(* CoDeSys 2.3 export: MIR_KOMPRESSOR.EXP *)

(* POU PLC_PRG, ST *)
PROGRAM PLC_PRG
VAR
	a : BOOL;
END_VAR
translate();
IF (_switchAuto) THEN
	work();
END_IF;
(*
start_or_stop(); *)
E_STOP();
END_PROGRAM

(* POU translate, ST *)
PROGRAM translate
VAR

	K3: BOOL;
	SC1: SCALE;
	SC2: SCALE;
	SC3: SCALE;
	SC4: SCALE;
	SC5: SCALE;
	SC6: SCALE;
	SC7: SCALE;
	SC8: SCALE;
	SC9: SCALE;
	SC10: SCALE;
	SC11: SCALE;
	SC12: SCALE;
END_VAR
MODBUS();
ANALOG();
K01 := TRM7;
K1 := _1pressLevelInDI;
K2 := _2pressLevelInDI;
K3 := _3pressLevelInDI;
K4 := _4pressLevelInDI;
 _rejimModeDO := P2;

IF (kompOnDO_MB = TRUE) THEN
	_kompOnDO :=  kompOnDO_MB;
ELSE
	_kompOnDO := FALSE;
END_IF;
IF (kompOffDO_MB = TRUE ) THEN
	_kompOffDO :=  kompOffDO_MB;
ELSE
	_kompOffDO := FALSE;
END_IF
END_PROGRAM
ACTION ANALOG:
SC1(IN := %IW0, MIN_VALUE := 4, MAX_VALUE := 20, OUT => analog1);
SC2(IN := %IW1, MIN_VALUE := 4, MAX_VALUE := 20, OUT => analog2);
SC3(IN := %IW2, MIN_VALUE := 4, MAX_VALUE := 20, OUT => analog3);
SC4(IN := %IW3, MIN_VALUE := 4, MAX_VALUE := 20, OUT => analog4);
SC5(IN := %IW4,MIN_VALUE := 4, MAX_VALUE := 20,  OUT => analog5);
SC6(IN := %IW5,MIN_VALUE := 4, MAX_VALUE := 20,  OUT => analog6);
SC7(IN := %IW6, MIN_VALUE := 4, MAX_VALUE := 20, OUT => analog7);
SC8(IN := %IW7, MIN_VALUE := 4, MAX_VALUE := 20, OUT => analog8);
SC9(IN := %IW8, MIN_VALUE := 4, MAX_VALUE := 20, OUT => analog9);
SC10(IN := %IW9, MIN_VALUE := 4, MAX_VALUE := 20, OUT => analog10);
SC11(IN := %IW10, MIN_VALUE := 4, MAX_VALUE := 20, OUT => analog11);
SC12(IN := %IW11, MIN_VALUE := 4, MAX_VALUE := 20, OUT => analog12);
END_ACTION
ACTION MODBUS:
S4_1MB := S4_1;
S4_2MB := S4_2;
S5_1MB := S5_1;
S5_2MB := S5_2;
S6_1MB := S6_1;
S6_2MB := S6_2;
S7_1MB := S7_1;
S7_2MB := S7_2;
S8_1MB := S8_1;
S8_2MB := S8_2;
S9_1MB := S9_1;
S9_2MB := S9_2;
S10_1MB := S10_1;
S10_2MB := S10_2;
S11_1MB := S11_1;
S11_2MB := S11_2;
S14_1MB := S14_1;
S14_2MB := S14_2;
S18_1MB := S18_1;
S18_2MB := S18_2;
S19_1MB := S19_1;
S19_2MB := S19_2;
controlFazaDIMB := _controlFazaDI;
currentHighJD5DIMB := _currentHighJD5DI;
vacumContactOnDIMB := _vacumContactOnDI;
press1LevelInDIMB := _1pressLevelInDI;
press2LevelInDIMB := _2pressLevelInDI;
press3LevelInDIMB := _3pressLevelInDI;
press4LevelInDIMB := _4pressLevelInDI;
press4LevelOutDIMB :=_4pressLeveOutDI;
pressWaterDIMB := _pressWaterDI;

KM4_1MB := KM4_1;
KM4_2MB := KM4_2;
KM5_1MB := KM5_1;
KM5_2MB := KM5_2;
KM6_1MB := KM6_1;
KM6_2MB := KM6_2;
KM7_1MB := KM7_1;
KM7_2MB := KM7_2;
KM8_1MB := KM8_1;
KM8_2MB := KM8_2;
KM9_1MB := KM9_1;
KM9_2MB := KM9_2;
KM10_1MB := KM10_1;
KM10_2MB := KM10_2;
KM11_1MB := KM11_1;
KM11_2MB := KM11_2;

KM14_1MB := KM14_1;
KM14_2MB := KM14_2;
KM18_1MB := KM18_1;
KM18_2MB := KM18_2;
KM19_1MB := KM19_1;
KM19_2MB := KM19_2;
KM1_MB := KM1;
KM2_MB := KM2;
(*
kompOnDO_MB := _kompOnDO;
kompOffDO_MB := _kompOffDO;*)
alarmLedDO_MB := _alarmLedDO;
stopModeDO_MB := _stopModeDO;

konsovikMechanikMotor := _konsovikMechanikMotor;
emergencyStop_MB := NOT _emergencyStop;
SBA41_MB := SBA41;
SB42_MB := SB42;
SB43_MB := SB43;
SB44_MB := SB44;
SB53_1MB := SB53_1;




buttonStop_MB := _buttonStop;
buttonRejim_MB := _buttonRejim;
buttonPusk_MB := _buttonPusk;
switchAuto_MB := _switchAuto;
switchManual_MB := _switchManual;
emergencyStopmashZal_MB := NOT  _emergencyStopMashZal;
END_ACTION

(* POU SCALE, ST *)
FUNCTION_BLOCK SCALE
VAR_INPUT
	IN : WORD;
	MIN_VALUE : REAL := 4;
	MAX_VALUE : REAL := 20;
END_VAR
VAR_OUTPUT
	OUT : REAL;
END_VAR
VAR
	T : REAL;
END_VAR
T := WORD_TO_REAL(IN);
OUT := (MAX_VALUE - MIN_VALUE) * T / 32767 +  MIN_VALUE;
END_FUNCTION_BLOCK

(* POU work, ST *)
PROGRAM work
VAR


END_VAR
	L05();
	L08();
	L09();
	L10();
	L11();
	L12();
	L13();
	L14();
	L15();
	L16();
END_PROGRAM

(* POU L05, CFC *)
PROGRAM L05
VAR
	_kompOffDO000000000: BOOL;
END_VAR
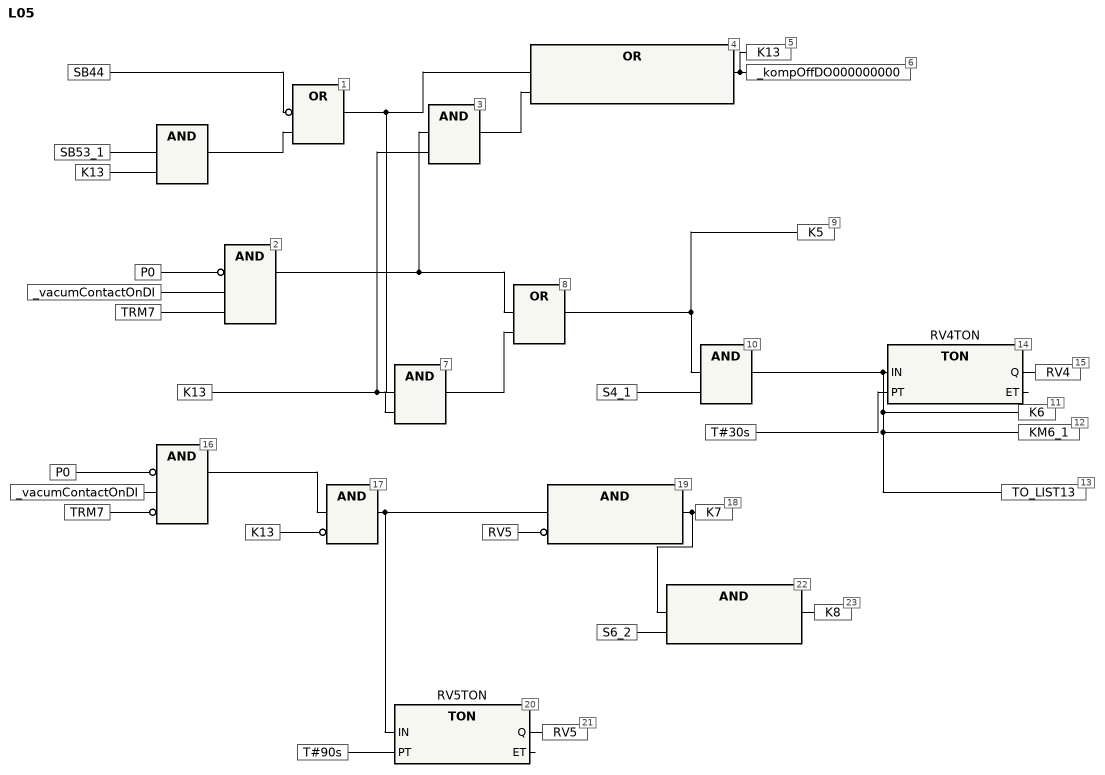
_CFC_ (* Continuous Function Chart, elements in execution order *)
#0 AND(SB53_1, K13)
#1 OR(NOT SB44, #0)
#2 AND(NOT P0, _vacumContactOnDI, TRM7)
#3 AND(#2, K13)
#4 OR(#1, #3)
#5 K13 <= #4
#6 _kompOffDO000000000 <= #4
#7 AND(#1, K13)
#8 OR(#2, #7)
#9 K5 <= #8
#10 AND(#8, S4_1)
#11 K6 <= #10
#12 KM6_1 <= #10
#13 TO_LIST13 <= #10
#14 RV4TON:TON(IN: #10, PT: T#30s)
#15 RV4 <= #14.Q
#16 AND(NOT P0, _vacumContactOnDI, NOT TRM7)
#17 AND(#16, NOT K13)
#18 K7 <= #19
#19 AND(#17, NOT RV5)
#20 RV5TON:TON(IN: #17, PT: T#90s)
#21 RV5 <= #20.Q
#22 AND(#19, S6_2)
#23 K8 <= #22
_END_CFC_
END_PROGRAM

(* POU L08, CFC *)
PROGRAM L08
VAR


END_VAR
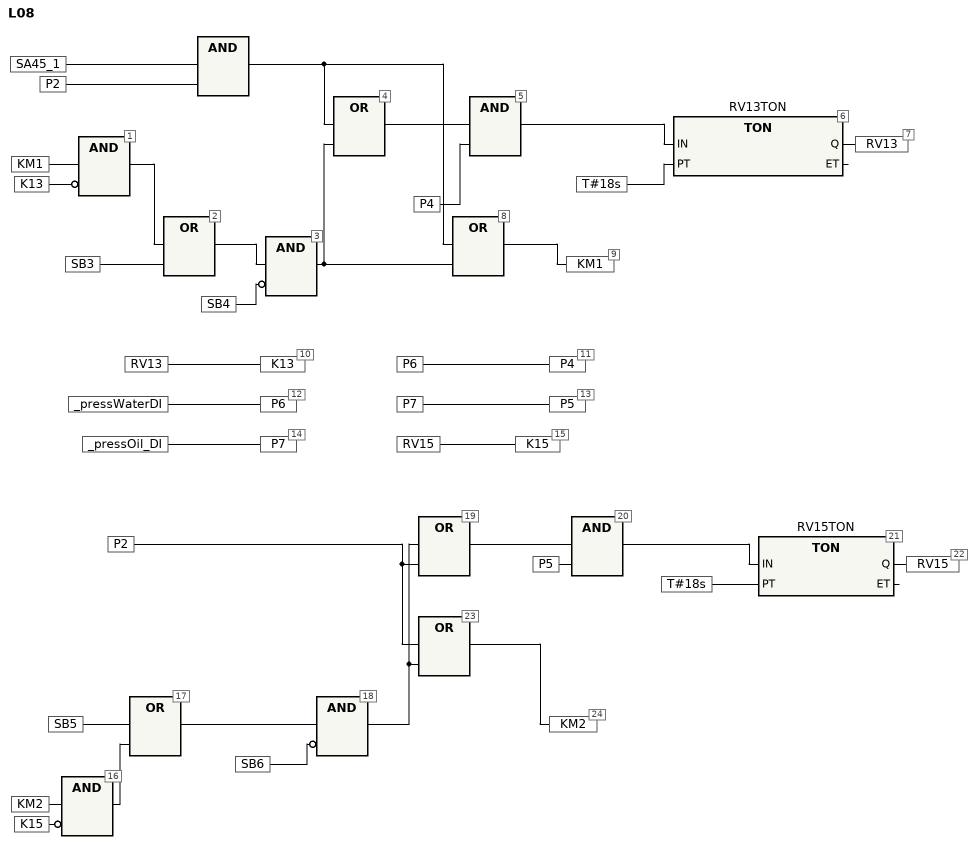
_CFC_ (* Continuous Function Chart, elements in execution order *)
#0 AND(SA45_1, P2)
#1 AND(KM1, NOT K13)
#2 OR(#1, SB3)
#3 AND(#2, NOT SB4)
#4 OR(#0, #3)
#5 AND(#4, P4)
#6 RV13TON:TON(IN: #5, PT: T#18s)
#7 RV13 <= #6.Q
#8 OR(#0, #3)
#9 KM1 <= #8
#10 K13 <= RV13
#11 P4 <= P6
#12 P6 <= _pressWaterDI
#13 P5 <= P7
#14 P7 <= _pressOil_DI
#15 K15 <= RV15
#16 AND(KM2, NOT K15)
#17 OR(SB5, #16)
#18 AND(#17, NOT SB6)
#19 OR(#18, P2)
#20 AND(#19, P5)
#21 RV15TON:TON(IN: #20, PT: T#18s)
#22 RV15 <= #21.Q
#23 OR(P2, #18)
#24 KM2 <= #23
_END_CFC_
END_PROGRAM

(* POU L09, CFC *)
PROGRAM L09
VAR




END_VAR
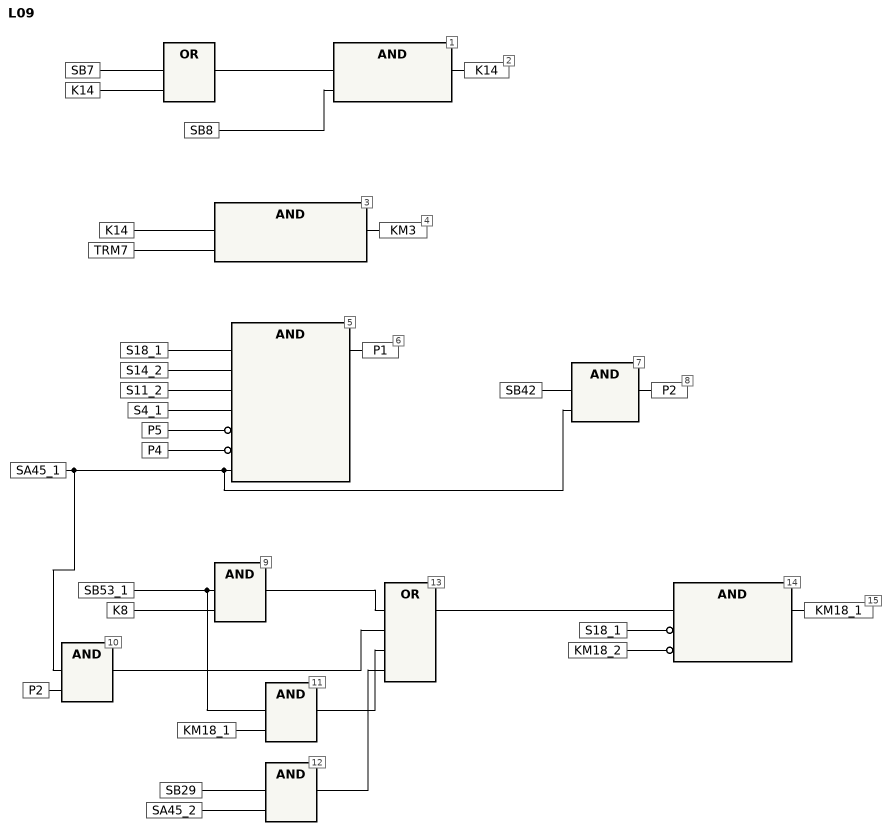
_CFC_ (* Continuous Function Chart, elements in execution order *)
#0 OR(SB7, K14)
#1 AND(#0, SB8)
#2 K14 <= #1
#3 AND(K14, TRM7)
#4 KM3 <= #3
#5 AND(S18_1, S14_2, S11_2, S4_1, NOT P5, NOT P4, SA45_1)
#6 P1 <= #5
#7 AND(SB42, SA45_1)
#8 P2 <= #7
#9 AND(SB53_1, K8)
#10 AND(SA45_1, P2)
#11 AND(SB53_1, KM18_1)
#12 AND(SB29, SA45_2)
#13 OR(#9, #10, #11, #12)
#14 AND(#13, NOT S18_1, NOT KM18_2)
#15 KM18_1 <= #14
_END_CFC_
(* the same logic as Structured Text *)
K14 := (SB7 OR K14) AND SB8;
KM3 := K14 AND TRM7;
P1 := S18_1 AND S14_2 AND S11_2 AND S4_1 AND NOT P5 AND NOT P4 AND SA45_1;
P2 := SB42 AND SA45_1;
KM18_1 := ((SB53_1 AND K8) OR (SA45_1 AND P2) OR (SB53_1 AND KM18_1) OR (SB29 AND SA45_2)) AND NOT S18_1 AND NOT KM18_2;
END_PROGRAM

(* POU L10, CFC *)
PROGRAM L10
VAR
	_17S_2: BOOL;
END_VAR
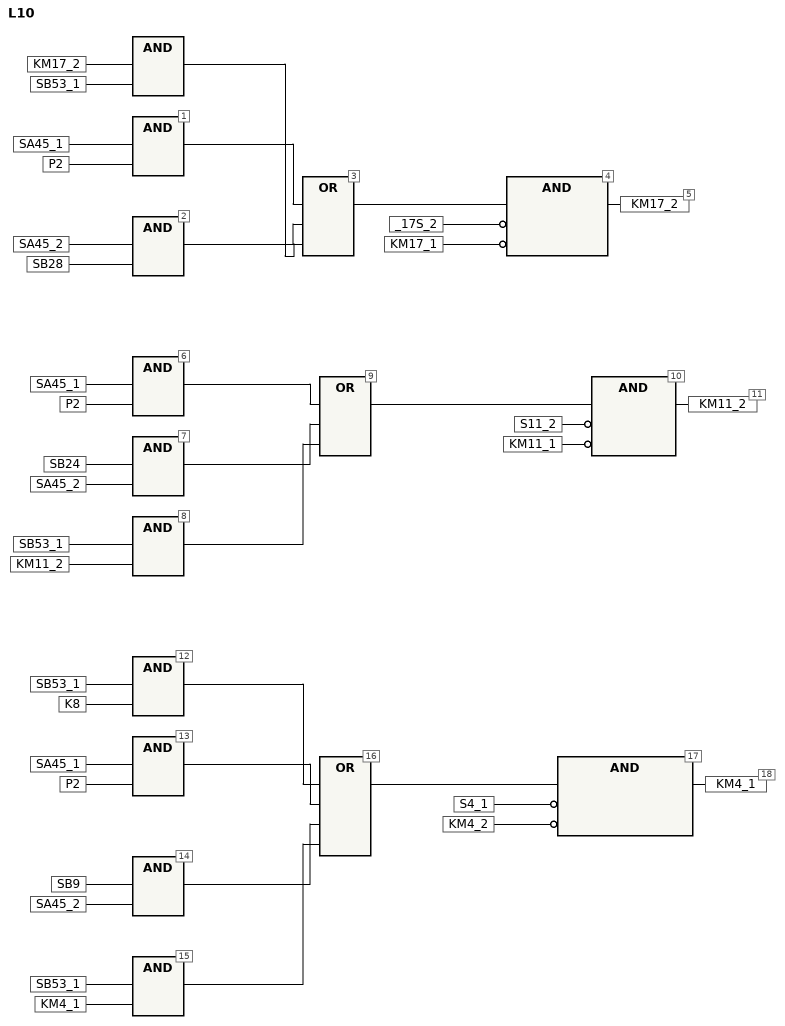
_CFC_ (* Continuous Function Chart, elements in execution order *)
#0 AND(KM17_2, SB53_1)
#1 AND(SA45_1, P2)
#2 AND(SA45_2, SB28)
#3 OR(#1, #2, #0)
#4 AND(#3, NOT _17S_2, NOT KM17_1)
#5 KM17_2 <= #4
#6 AND(SA45_1, P2)
#7 AND(SB24, SA45_2)
#8 AND(SB53_1, KM11_2)
#9 OR(#6, #7, #8)
#10 AND(#9, NOT S11_2, NOT KM11_1)
#11 KM11_2 <= #10
#12 AND(SB53_1, K8)
#13 AND(SA45_1, P2)
#14 AND(SB9, SA45_2)
#15 AND(SB53_1, KM4_1)
#16 OR(#12, #13, #14, #15)
#17 AND(#16, NOT S4_1, NOT KM4_2)
#18 KM4_1 <= #17
_END_CFC_
(* the same logic as Structured Text *)
KM17_2 := ((SA45_1 AND P2) OR (SA45_2 AND SB28) OR (KM17_2 AND SB53_1)) AND NOT _17S_2 AND NOT KM17_1;
KM11_2 := ((SA45_1 AND P2) OR (SB24 AND SA45_2) OR (SB53_1 AND KM11_2)) AND NOT S11_2 AND NOT KM11_1;
KM4_1 := ((SB53_1 AND K8) OR (SA45_1 AND P2) OR (SB9 AND SA45_2) OR (SB53_1 AND KM4_1)) AND NOT S4_1 AND NOT KM4_2;
END_PROGRAM

(* POU L11, CFC *)
PROGRAM L11
VAR


	_16S_2: BOOL;
END_VAR
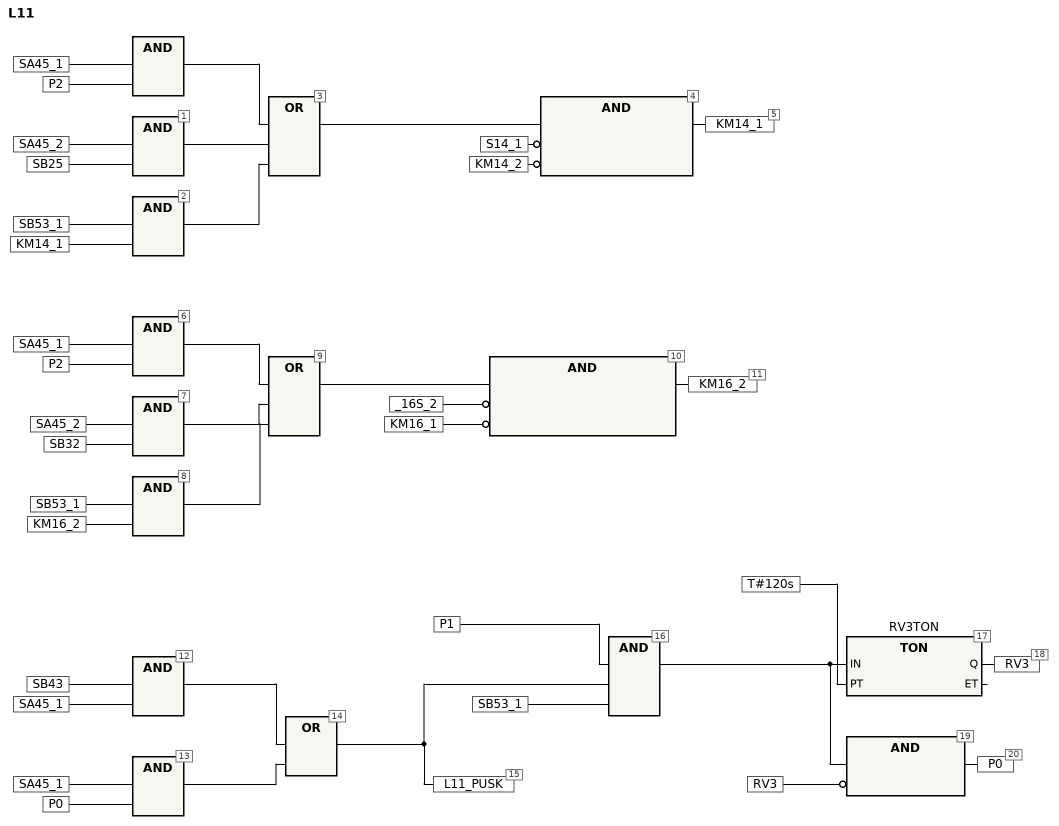
_CFC_ (* Continuous Function Chart, elements in execution order *)
#0 AND(SA45_1, P2)
#1 AND(SA45_2, SB25)
#2 AND(SB53_1, KM14_1)
#3 OR(#0, #1, #2)
#4 AND(#3, NOT S14_1, NOT KM14_2)
#5 KM14_1 <= #4
#6 AND(SA45_1, P2)
#7 AND(SA45_2, SB32)
#8 AND(SB53_1, KM16_2)
#9 OR(#6, #7, #8)
#10 AND(#9, NOT _16S_2, NOT KM16_1)
#11 KM16_2 <= #10
#12 AND(SB43, SA45_1)
#13 AND(SA45_1, P0)
#14 OR(#12, #13)
#15 L11_PUSK <= #14
#16 AND(P1, #14, SB53_1)
#17 RV3TON:TON(IN: #16, PT: T#120s)
#18 RV3 <= #17.Q
#19 AND(#16, NOT RV3)
#20 P0 <= #19
_END_CFC_
END_PROGRAM

(* POU L12, CFC *)
PROGRAM L12
VAR







END_VAR
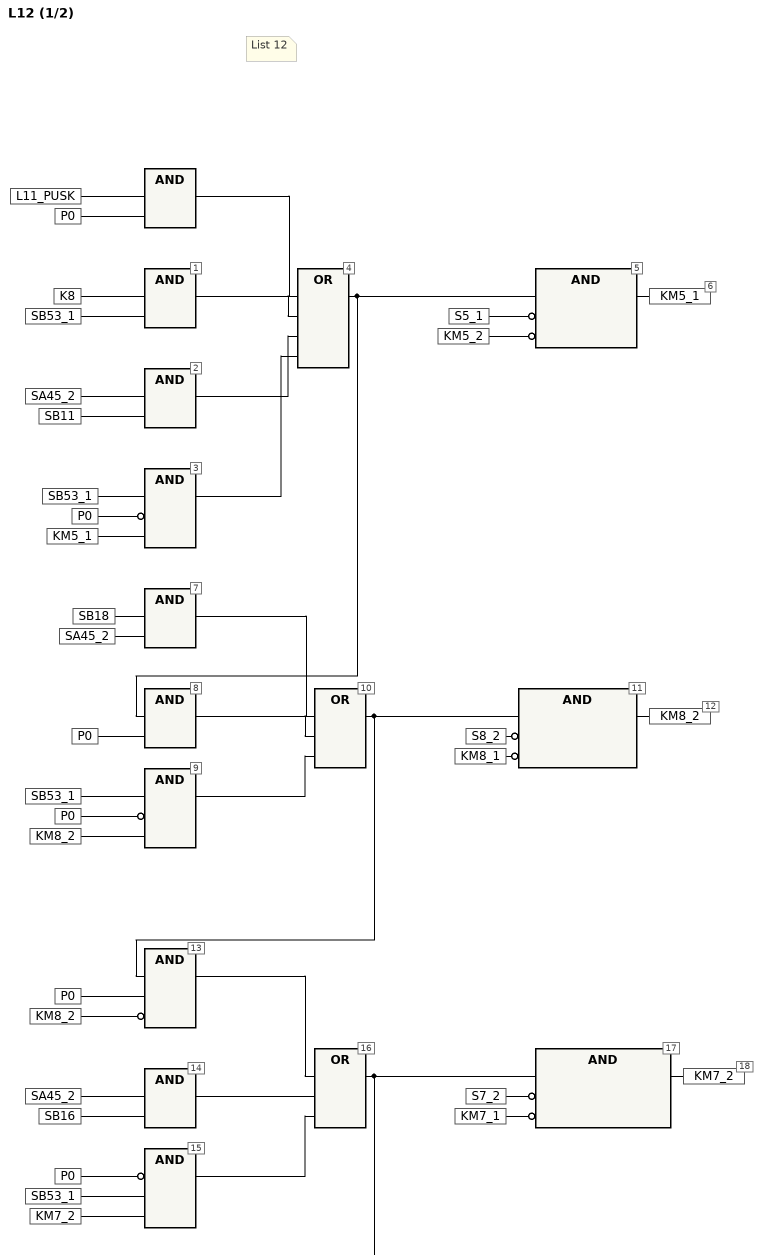
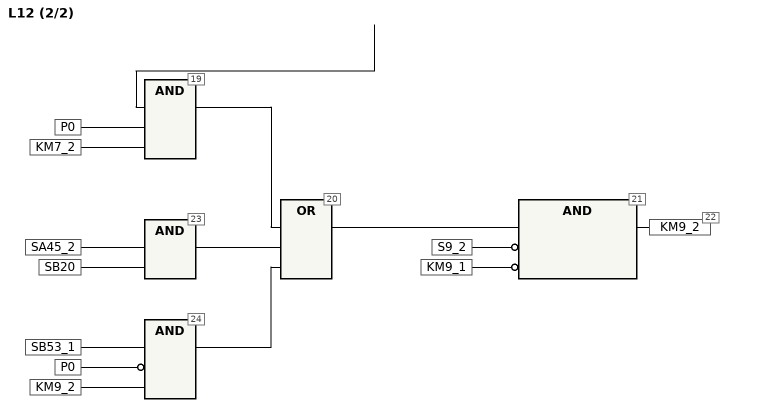
_CFC_ (* Continuous Function Chart, elements in execution order *)
(* List 12 *)
#0 AND(L11_PUSK, P0)
#1 AND(K8, SB53_1)
#2 AND(SA45_2, SB11)
#3 AND(SB53_1, NOT P0, KM5_1)
#4 OR(#0, #1, #2, #3)
#5 AND(#4, NOT S5_1, NOT KM5_2)
#6 KM5_1 <= #5
#7 AND(SB18, SA45_2)
#8 AND(#4, P0)
#9 AND(SB53_1, NOT P0, KM8_2)
#10 OR(#7, #8, #9)
#11 AND(#10, NOT S8_2, NOT KM8_1)
#12 KM8_2 <= #11
#13 AND(#10, P0, NOT KM8_2)
#14 AND(SA45_2, SB16)
#15 AND(NOT P0, SB53_1, KM7_2)
#16 OR(#13, #14, #15)
#17 AND(#16, NOT S7_2, NOT KM7_1)
#18 KM7_2 <= #17
#19 AND(#16, P0, KM7_2)
#20 OR(#19, #23, #24)
#21 AND(#20, NOT S9_2, NOT KM9_1)
#22 KM9_2 <= #21
#23 AND(SA45_2, SB20)
#24 AND(SB53_1, NOT P0, KM9_2)
_END_CFC_
END_PROGRAM

(* POU L13, CFC *)
PROGRAM L13
VAR



	P4: BOOL;

END_VAR
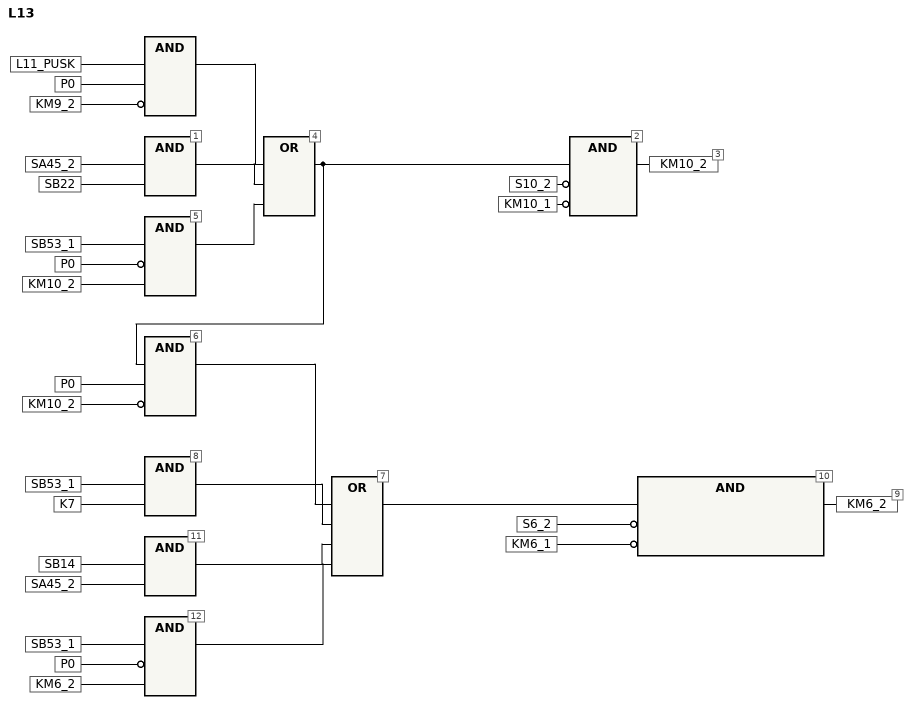
_CFC_ (* Continuous Function Chart, elements in execution order *)
#0 AND(L11_PUSK, P0, NOT KM9_2)
#1 AND(SA45_2, SB22)
#2 AND(#4, NOT S10_2, NOT KM10_1)
#3 KM10_2 <= #2
#4 OR(#0, #1, #5)
#5 AND(SB53_1, NOT P0, KM10_2)
#6 AND(#4, P0, NOT KM10_2)
#7 OR(#6, #8, #11, #12)
#8 AND(SB53_1, K7)
#9 KM6_2 <= #10
#10 AND(#7, NOT S6_2, NOT KM6_1)
#11 AND(SB14, SA45_2)
#12 AND(SB53_1, NOT P0, KM6_2)
_END_CFC_
END_PROGRAM

(* POU L14, CFC *)
PROGRAM L14
VAR

END_VAR
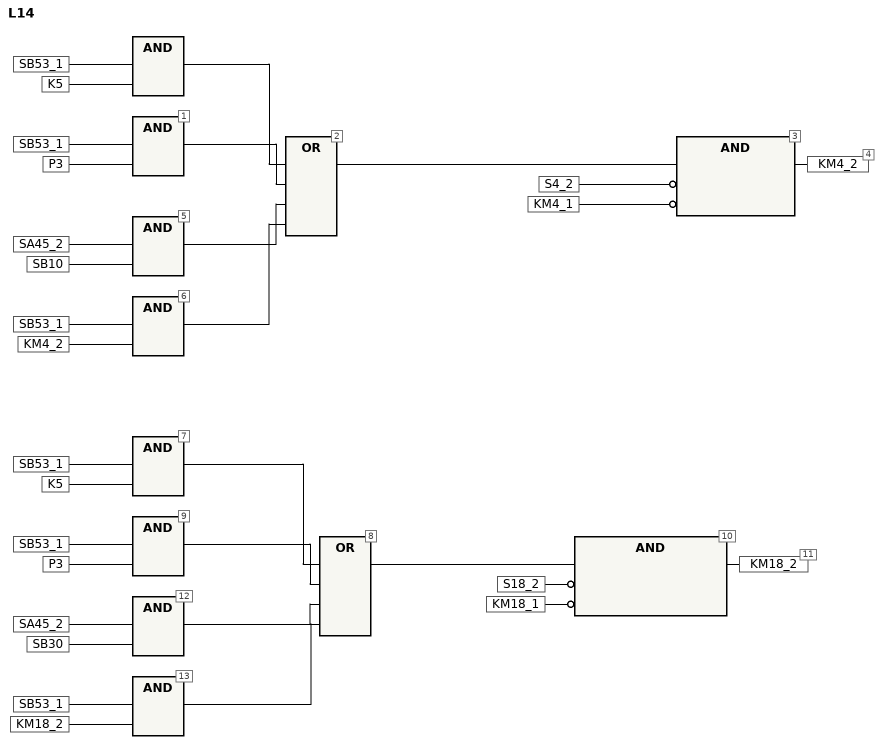
_CFC_ (* Continuous Function Chart, elements in execution order *)
#0 AND(SB53_1, K5)
#1 AND(SB53_1, P3)
#2 OR(#0, #1, #5, #6)
#3 AND(#2, NOT S4_2, NOT KM4_1)
#4 KM4_2 <= #3
#5 AND(SA45_2, SB10)
#6 AND(SB53_1, KM4_2)
#7 AND(SB53_1, K5)
#8 OR(#7, #9, #12, #13)
#9 AND(SB53_1, P3)
#10 AND(#8, NOT S18_2, NOT KM18_1)
#11 KM18_2 <= #10
#12 AND(SA45_2, SB30)
#13 AND(SB53_1, KM18_2)
_END_CFC_
END_PROGRAM

(* POU L15, CFC *)
PROGRAM L15
VAR

END_VAR
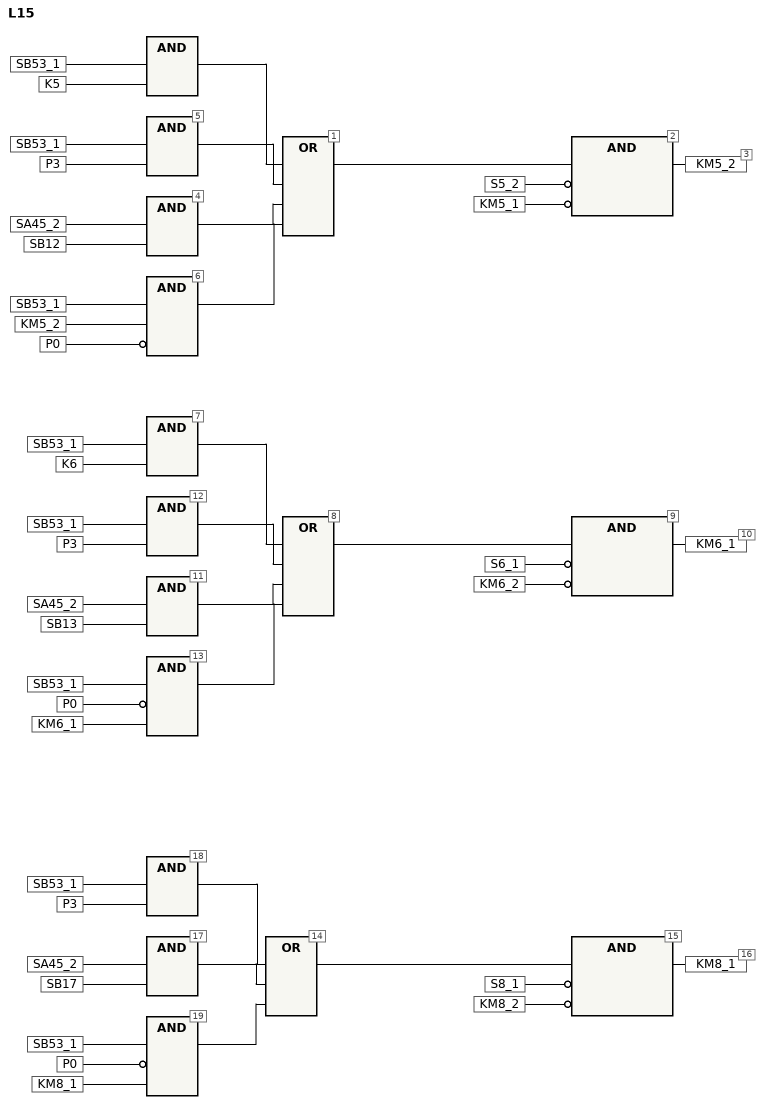
_CFC_ (* Continuous Function Chart, elements in execution order *)
#0 AND(SB53_1, K5)
#1 OR(#0, #5, #4, #6)
#2 AND(#1, NOT S5_2, NOT KM5_1)
#3 KM5_2 <= #2
#4 AND(SA45_2, SB12)
#5 AND(SB53_1, P3)
#6 AND(SB53_1, KM5_2, NOT P0)
#7 AND(SB53_1, K6)
#8 OR(#7, #12, #11, #13)
#9 AND(#8, NOT S6_1, NOT KM6_2)
#10 KM6_1 <= #9
#11 AND(SA45_2, SB13)
#12 AND(SB53_1, P3)
#13 AND(SB53_1, NOT P0, KM6_1)
#14 OR(#18, #17, #19)
#15 AND(#14, NOT S8_1, NOT KM8_2)
#16 KM8_1 <= #15
#17 AND(SA45_2, SB17)
#18 AND(SB53_1, P3)
#19 AND(SB53_1, NOT P0, KM8_1)
_END_CFC_
END_PROGRAM

(* POU L16, CFC *)
PROGRAM L16
VAR





END_VAR
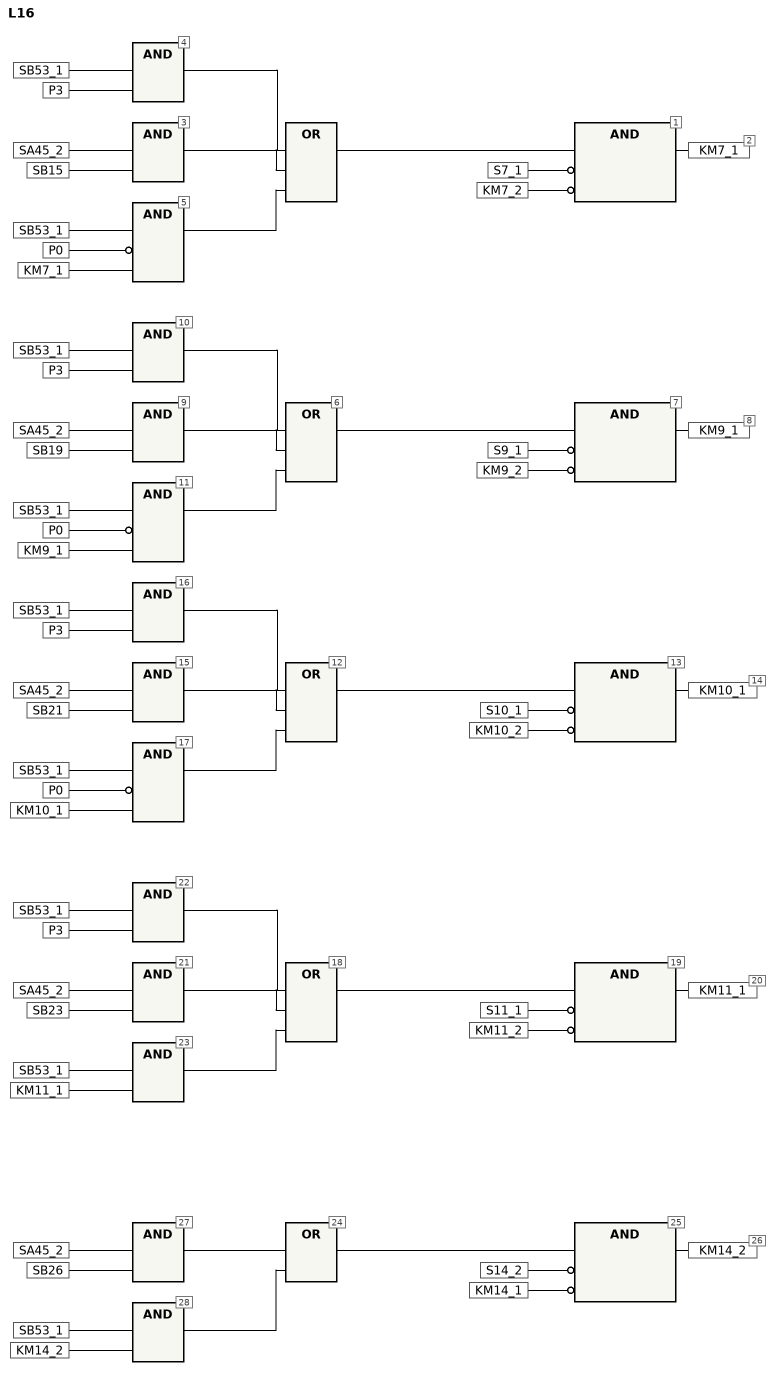
_CFC_ (* Continuous Function Chart, elements in execution order *)
#0 OR(#4, #3, #5)
#1 AND(#0, NOT S7_1, NOT KM7_2)
#2 KM7_1 <= #1
#3 AND(SA45_2, SB15)
#4 AND(SB53_1, P3)
#5 AND(SB53_1, NOT P0, KM7_1)
#6 OR(#10, #9, #11)
#7 AND(#6, NOT S9_1, NOT KM9_2)
#8 KM9_1 <= #7
#9 AND(SA45_2, SB19)
#10 AND(SB53_1, P3)
#11 AND(SB53_1, NOT P0, KM9_1)
#12 OR(#16, #15, #17)
#13 AND(#12, NOT S10_1, NOT KM10_2)
#14 KM10_1 <= #13
#15 AND(SA45_2, SB21)
#16 AND(SB53_1, P3)
#17 AND(SB53_1, NOT P0, KM10_1)
#18 OR(#22, #21, #23)
#19 AND(#18, NOT S11_1, NOT KM11_2)
#20 KM11_1 <= #19
#21 AND(SA45_2, SB23)
#22 AND(SB53_1, P3)
#23 AND(SB53_1, KM11_1)
#24 OR(#27, #28)
#25 AND(#24, NOT S14_2, NOT KM14_1)
#26 KM14_2 <= #25
#27 AND(SA45_2, SB26)
#28 AND(SB53_1, KM14_2)
_END_CFC_
END_PROGRAM

(* POU E_STOP, LD *)
PROGRAM E_STOP
VAR



	P4: BOOL;

	trig: R_TRIG;
END_VAR
VAR
	_ImpVar_78_35:	BOOL;
	_ImpVar_78_38:	BOOL;

END_VAR
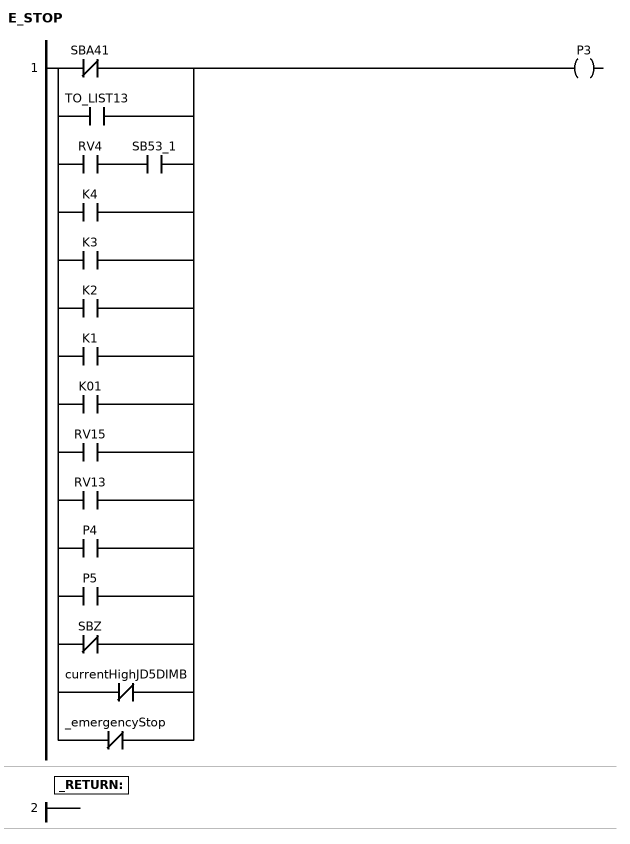
_LD_ (* Ladder Diagram *)
NETWORK 1
	{ [/SBA41] | [TO_LIST13] | [RV4] - [SB53_1] | [K4] | [K3] | [K2] | [K1] | [K01] | [RV15] | [RV13] | [P4] | [P5] | [/SBZ] | [/currentHighJD5DIMB] | [/_emergencyStop] } --- (P3)
NETWORK 2 _RETURN::
	*
_END_LD_
(* the same logic as Structured Text *)
(* Network 1 *)
P3 := NOT SBA41 OR TO_LIST13 OR RV4 AND SB53_1 OR K4 OR K3 OR K2 OR K1 OR K01 OR RV15 OR RV13 OR P4 OR P5 OR NOT SBZ OR NOT currentHighJD5DIMB OR NOT _emergencyStop;
(* Network 2 *)
(* label: _RETURN: *)
END_PROGRAM

(* POU list5, LD *)
PROGRAM list5
VAR
	stopKomp: BOOL;
	stopZadv: BOOL;
	k13: BOOL;
	tempK13: BOOL;
	K5: BOOL;
	P0: BOOL;
	TRM7: BOOL;
	VV: BOOL;
	tempTRM7: BOOL;
	RV4: BOOL;
	tempRV4: BOOL;
	RV4TON: TON;
END_VAR
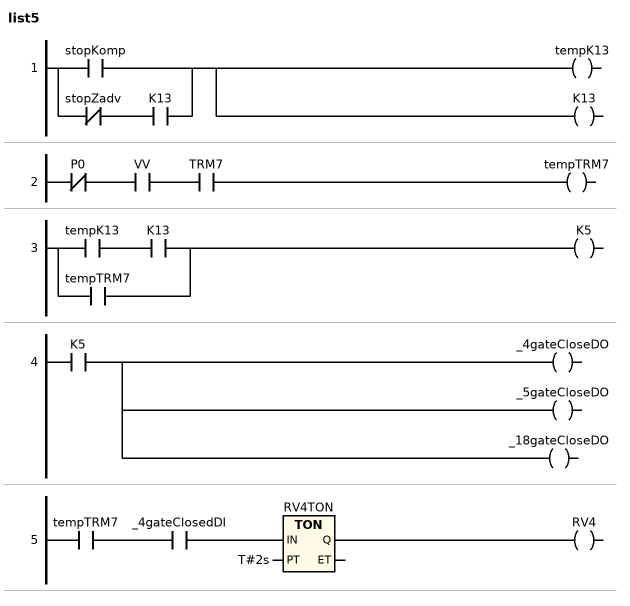
_LD_ (* Ladder Diagram *)
NETWORK 1
	{ [stopKomp] | [/stopZadv] - [K13] } --- (tempK13) (K13)
NETWORK 2
	[/P0] - [VV] - [TRM7] --- (tempTRM7)
NETWORK 3
	{ [tempK13] - [K13] | [tempTRM7] } --- (K5)
NETWORK 4
	[K5] --- (_4gateCloseDO) (_5gateCloseDO) (_18gateCloseDO)
NETWORK 5
	[tempTRM7] - [_4gateClosedDI] - RV4TON:TON(IN: *, PT: T#2s) --- (RV4)
_END_LD_
(* the same logic as Structured Text *)
(* Network 1 *)
tempK13 := stopKomp OR NOT stopZadv AND K13;
K13 := tempK13;
(* Network 2 *)
tempTRM7 := NOT P0 AND VV AND TRM7;
(* Network 3 *)
K5 := tempK13 AND K13 OR tempTRM7;
(* Network 4 *)
_4gateCloseDO := K5;
_5gateCloseDO := K5;
_18gateCloseDO := K5;
(* Network 5 *)
RV4TON(IN := tempTRM7 AND _4gateClosedDI, PT := T#2s);
RV4 := RV4TON.Q;
END_PROGRAM

(* POU nur, LD *)
PROGRAM nur
VAR
	rejim : BOOL;
	pusk: BOOL;
END_VAR
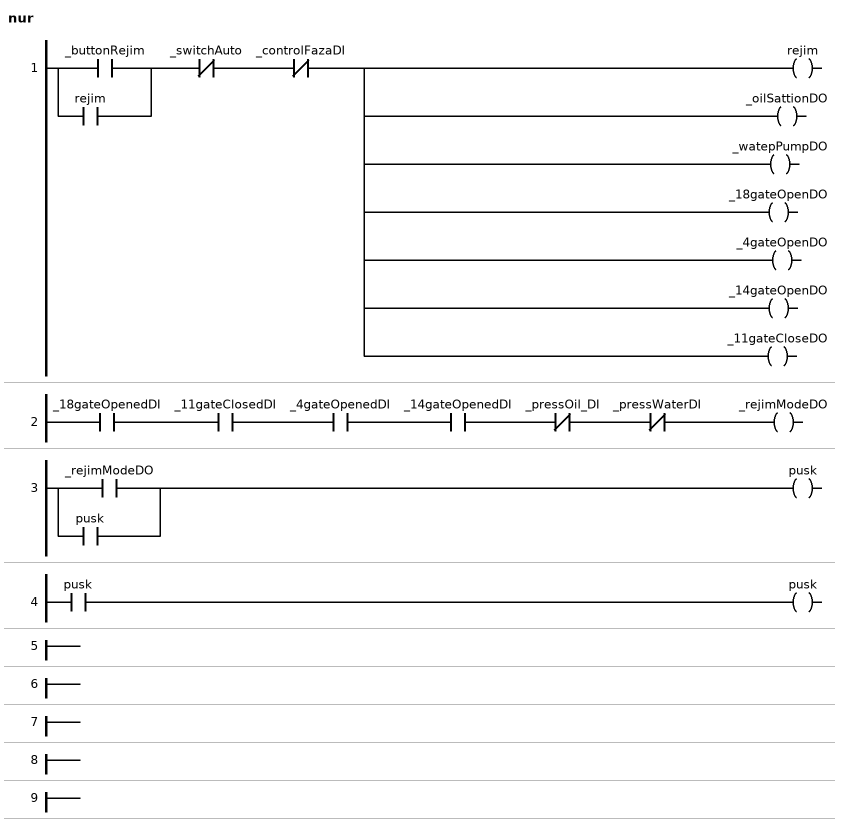
_LD_ (* Ladder Diagram *)
NETWORK 1
	{ [_buttonRejim] | [rejim] } - [/_switchAuto] - [/_controlFazaDI] --- (rejim) (_oilSattionDO) (_watepPumpDO) (_18gateOpenDO) (_4gateOpenDO) (_14gateOpenDO) (_11gateCloseDO)
NETWORK 2
	[_18gateOpenedDI] - [_11gateClosedDI] - [_4gateOpenedDI] - [_14gateOpenedDI] - [/_pressOil_DI] - [/_pressWaterDI] --- (_rejimModeDO)
NETWORK 3
	{ [_rejimModeDO] | [pusk] } --- (pusk)
NETWORK 4
	[pusk] --- (pusk)
NETWORK 5
	*
NETWORK 6
	*
NETWORK 7
	*
NETWORK 8
	*
NETWORK 9
	*
_END_LD_
(* the same logic as Structured Text *)
(* Network 1 *)
rejim := (_buttonRejim OR rejim) AND NOT _switchAuto AND NOT _controlFazaDI;
_oilSattionDO := rejim;
_watepPumpDO := rejim;
_18gateOpenDO := rejim;
_4gateOpenDO := rejim;
_14gateOpenDO := rejim;
_11gateCloseDO := rejim;
(* Network 2 *)
_rejimModeDO := _18gateOpenedDI AND _11gateClosedDI AND _4gateOpenedDI AND _14gateOpenedDI AND NOT _pressOil_DI AND NOT _pressWaterDI;
(* Network 3 *)
pusk := _rejimModeDO OR pusk;
(* Network 4 *)
pusk := pusk;
(* Network 5 *)
(* Network 6 *)
(* Network 7 *)
(* Network 8 *)
(* Network 9 *)
END_PROGRAM

(* POU start_or_stop, LD *)
PROGRAM start_or_stop
VAR
	_controlFazaDI46: BOOL;
	kompressorOFF: TP;
	kompressorON: TP;
	_currentHighJD5DI00000: BOOL;
	P300000: BOOL;
	P00000: BOOL;
	trig: R_TRIG;
	alarmLedDO_MB555: BOOL;
END_VAR
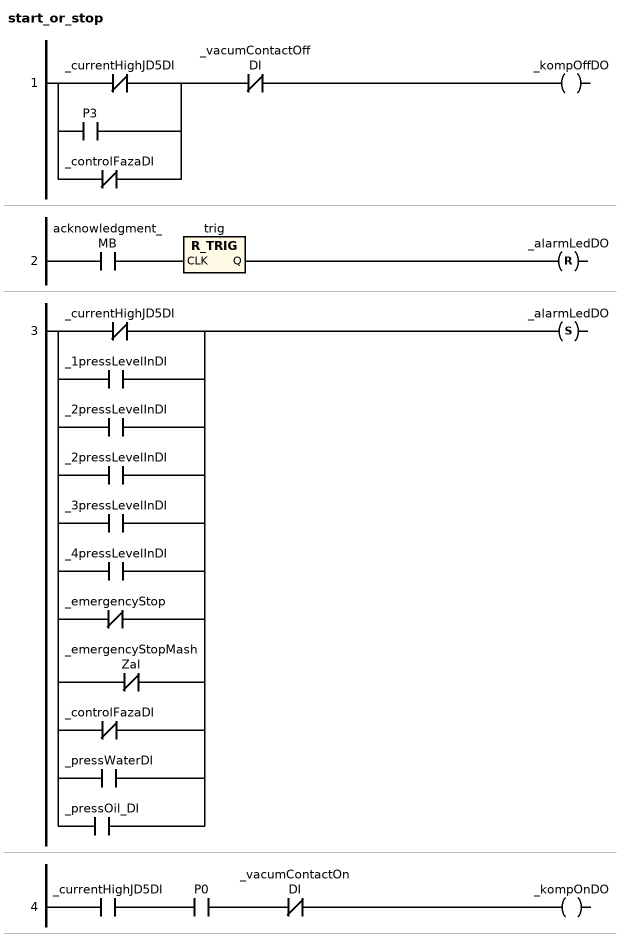
_LD_ (* Ladder Diagram *)
NETWORK 1
	{ [/_currentHighJD5DI] | [P3] | [/_controlFazaDI] } - [/_vacumContactOffDI] --- (_kompOffDO)
NETWORK 2
	[acknowledgment_MB] - trig:R_TRIG(CLK: *) --- (R _alarmLedDO)
NETWORK 3
	{ [/_currentHighJD5DI] | [_1pressLevelInDI] | [_2pressLevelInDI] | [_2pressLevelInDI] | [_3pressLevelInDI] | [_4pressLevelInDI] | [/_emergencyStop] | [/_emergencyStopMashZal] | [/_controlFazaDI] | [_pressWaterDI] | [_pressOil_DI] } --- (S _alarmLedDO)
NETWORK 4
	[_currentHighJD5DI] - [P0] - [/_vacumContactOnDI] --- (_kompOnDO)
_END_LD_
(* the same logic as Structured Text *)
(* Network 1 *)
_kompOffDO := (NOT _currentHighJD5DI OR P3 OR NOT _controlFazaDI) AND NOT _vacumContactOffDI;
(* Network 2 *)
trig(CLK := acknowledgment_MB);
IF trig.Q THEN _alarmLedDO := FALSE; END_IF;
(* Network 3 *)
IF NOT _currentHighJD5DI OR _1pressLevelInDI OR _2pressLevelInDI OR _2pressLevelInDI OR _3pressLevelInDI OR _4pressLevelInDI OR NOT _emergencyStop OR NOT _emergencyStopMashZal OR NOT _controlFazaDI OR _pressWaterDI OR _pressOil_DI THEN _alarmLedDO := TRUE; END_IF;
(* Network 4 *)
_kompOnDO := _currentHighJD5DI AND P0 AND NOT _vacumContactOnDI;
END_PROGRAM
